// Device/Application/PLC_VISU
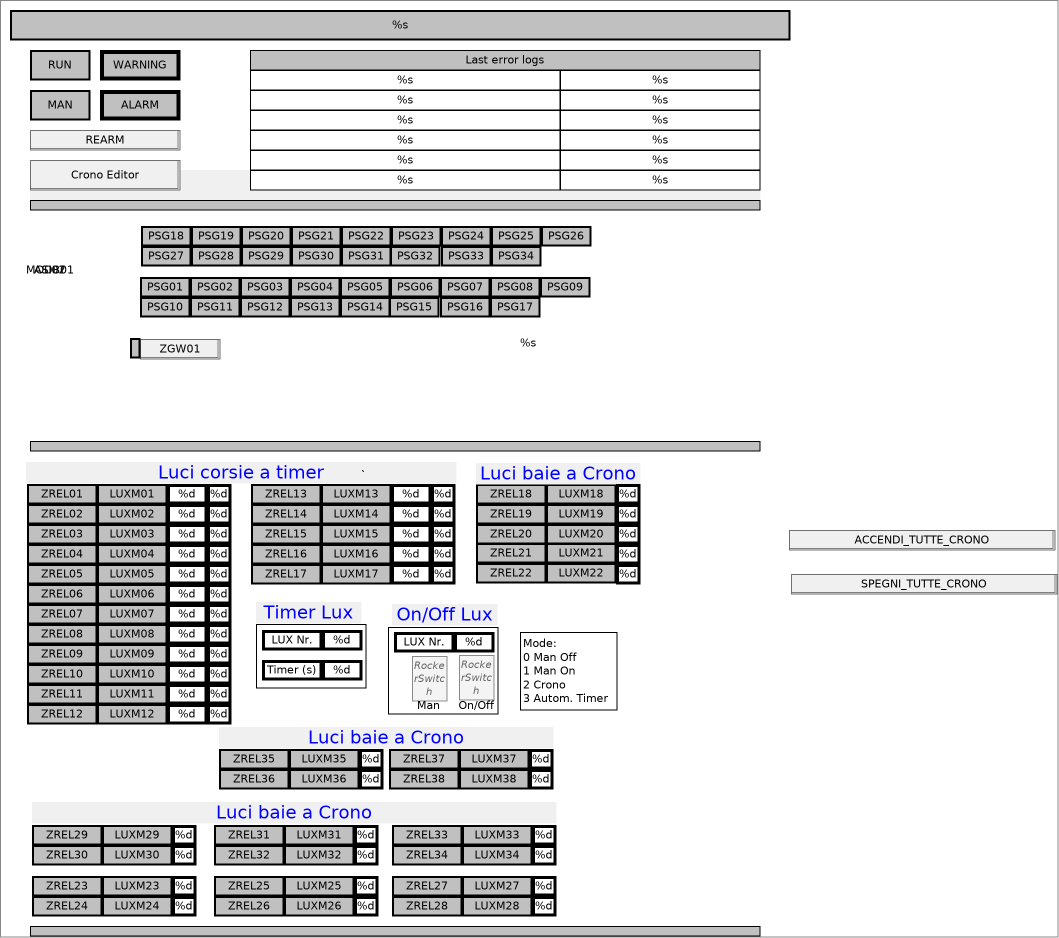
VISUALIZATION PLC_VISU  // 1059x938
    Rectangle (10,10 780x30), "%s", text variable: Plant_NAME
    Rectangle (30,441 730x10)
    Rectangle (30,170 730x30)
    Rectangle (30,926 730x10)
    Rectangle (30,200 730x10)
    Rectangle (319,333 220x20), "%s", text variable: Sys.Time_LogString
    Polygon (50,270), "MODB01", colour variable: MODB01.Status_Vis
    RoundedRectangle (30,50 60x30), "RUN", colour toggle: NOT Mode_Manual
        OnMouseUp: execute { Mode_Manual:=(FALSE); }
    RoundedRectangle (30,90 60x30), "MAN", colour toggle: Mode_Manual
        OnMouseUp: execute { Mode_Manual:=(TRUE); }
    Button (30,160 150x30), "Crono Editor"
        OnMouseUp:  Assign=VIS_CHONOEDITOR, Assign=VIS_CHONOEDITOR, Type=Assignment
    Rectangle (560,70 200x20), "%s", text variable: SYS.LastLogs_Msg[0]
    Polygon (240,190), invisible if: SYS.LastLogs_Idx<>0
    Rectangle (560,90 200x20), "%s", text variable: SYS.LastLogs_Msg[1]
    Polygon (240,90), invisible if: SYS.LastLogs_Idx<>1
    Rectangle (560,110 200x20), "%s", text variable: SYS.LastLogs_Msg[2]
    Polygon (240,110), invisible if: SYS.LastLogs_Idx<>2
    Rectangle (560,130 200x20), "%s", text variable: SYS.LastLogs_Msg[3]
    Polygon (240,130), invisible if: SYS.LastLogs_Idx<>3
    Rectangle (560,150 200x20), "%s", text variable: SYS.LastLogs_Msg[4]
    Polygon (240,150), invisible if: SYS.LastLogs_Idx<>4
    Rectangle (560,170 200x20), "%s", text variable: SYS.LastLogs_Msg[5]
    Polygon (240,170), invisible if: SYS.LastLogs_Idx<>5
    Rectangle (250,70 310x20), "%s", text variable: SYS.LastLogs_Dat[0]
    Rectangle (250,90 310x20), "%s", text variable: SYS.LastLogs_Dat[1]
    Rectangle (250,110 310x20), "%s", text variable: SYS.LastLogs_Dat[2]
    Rectangle (250,130 310x20), "%s", text variable: SYS.LastLogs_Dat[3]
    Rectangle (250,150 310x20), "%s", text variable: SYS.LastLogs_Dat[4]
    Rectangle (250,170 310x20), "%s", text variable: SYS.LastLogs_Dat[5]
    Rectangle (100,90 80x30), "ALARM", colour toggle: SYS.Alarm
    Rectangle (100,50 80x30), "WARNING", colour toggle: SYS.Warning
    Button (30,130 150x20), "REARM"
        OnMouseUp: execute { SYS.Alarm:=(FALSE); }
        OnMouseUp: execute { SYS.Warning:=(FALSE); }
    Rectangle (250,50 510x20), "Last error logs"
    Polygon (50,270), "ASI01", colour variable: ASI01.Status_Vis
    Polygon (50,270), "ASI02", colour variable: ASI02.Status_Vis
    Button (140,339 80x20), "ZGW01"
    Rectangle (130,338 10x20), colour variable: ZGW01.Status_Vis
    Line (130,246)
    Rectangle (140,297 50x20), "PSG10", colour variable: PSG[10].Status_Vis
    Rectangle (190,297 50x20), "PSG11", colour variable: PSG[11].Status_Vis
    Rectangle (240,297 50x20), "PSG12", colour variable: PSG[12].Status_Vis
    Rectangle (290,297 50x20), "PSG13", colour variable: PSG[13].Status_Vis
    Rectangle (219,769 70x20), "ZREL36", colour variable: ZREL[36].Status_Vis
    Rectangle (289,769 70x20), "LUXM36", colour variable: LUXM[36].Status_Vis
    Rectangle (219,749 70x20), "ZREL35", colour variable: ZREL[35].Status_Vis
    Rectangle (289,749 70x20), "LUXM35", colour variable: LUXM[35].Status_Vis
    Rectangle (389,769 70x20), "ZREL38", colour variable: ZREL[38].Status_Vis
    Rectangle (459,769 70x20), "LUXM38", colour variable: LUXM[38].Status_Vis
    Rectangle (389,749 70x20), "ZREL37", colour variable: ZREL[37].Status_Vis
    Rectangle (459,749 70x20), "LUXM37", colour variable: LUXM[37].Status_Vis
    Rectangle (219,727 334x21), "Luci baie a Crono"
    Rectangle (476,484 70x20), "ZREL18", colour variable: ZREL[18].Status_Vis
    Rectangle (476,504 70x20), "ZREL19", colour variable: ZREL[19].Status_Vis
    Rectangle (476,524 70x20), "ZREL20", colour variable: ZREL[20].Status_Vis
    Rectangle (476,543 70x20), "ZREL21", colour variable: ZREL[21].Status_Vis
    Rectangle (476,563 70x20), "ZREL22", colour variable: ZREL[22].Status_Vis
    Group (546,484 70x99)
        Rectangle (0,0 70x20), "LUXM18", colour variable: LUXM[18].Status_Vis
        Rectangle (0,20 70x20), "LUXM19", colour variable: LUXM[19].Status_Vis
        Rectangle (0,40 70x20), "LUXM20", colour variable: LUXM[20].Status_Vis
        Rectangle (0,59 70x20), "LUXM21", colour variable: LUXM[21].Status_Vis
        Rectangle (0,79 70x20), "LUXM22", colour variable: LUXM[22].Status_Vis
    Rectangle (476,463 164x21), "Luci baie a Crono"
    Rectangle (32,896 70x20), "ZREL24", colour variable: ZREL[24].Status_Vis
    Rectangle (102,896 70x20), "LUXM24", colour variable: LUXM[24].Status_Vis
    Rectangle (32,876 70x20), "ZREL23", colour variable: ZREL[23].Status_Vis
    Rectangle (102,876 70x20), "LUXM23", colour variable: LUXM[23].Status_Vis
    Rectangle (214,896 70x20), "ZREL26", colour variable: ZREL[26].Status_Vis
    Rectangle (284,896 70x20), "LUXM26", colour variable: LUXM[26].Status_Vis
    Rectangle (214,876 70x20), "ZREL25", colour variable: ZREL[25].Status_Vis
    Rectangle (284,876 70x20), "LUXM25", colour variable: LUXM[25].Status_Vis
    Rectangle (392,896 70x20), "ZREL28", colour variable: ZREL[28].Status_Vis
    Rectangle (462,896 70x20), "LUXM28", colour variable: LUXM[28].Status_Vis
    Rectangle (392,876 70x20), "ZREL27", colour variable: ZREL[27].Status_Vis
    Rectangle (462,876 70x20), "LUXM27", colour variable: LUXM[27].Status_Vis
    Rectangle (32,845 70x20), "ZREL30", colour variable: ZREL[30].Status_Vis
    Rectangle (102,845 70x20), "LUXM30", colour variable: LUXM[30].Status_Vis
    Rectangle (32,825 70x20), "ZREL29", colour variable: ZREL[29].Status_Vis
    Rectangle (102,825 70x20), "LUXM29", colour variable: LUXM[29].Status_Vis
    Rectangle (214,845 70x20), "ZREL32", colour variable: ZREL[32].Status_Vis
    Rectangle (284,845 70x20), "LUXM32", colour variable: LUXM[32].Status_Vis
    Rectangle (214,825 70x20), "ZREL31", colour variable: ZREL[31].Status_Vis
    Rectangle (284,825 70x20), "LUXM31", colour variable: LUXM[31].Status_Vis
    Rectangle (392,845 70x20), "ZREL34", colour variable: ZREL[34].Status_Vis
    Rectangle (462,845 70x20), "LUXM34", colour variable: LUXM[34].Status_Vis
    Rectangle (392,825 70x20), "ZREL33", colour variable: ZREL[33].Status_Vis
    Rectangle (462,825 70x20), "LUXM33", colour variable: LUXM[33].Status_Vis
    Rectangle (32,802 524x21), "Luci baie a Crono"
    Rectangle (340,297 50x20), "PSG14", colour variable: PSG[14].Status_Vis
    Rectangle (140,277 50x20), "PSG01", colour variable: PSG[1].Status_Vis
    Rectangle (190,277 50x20), "PSG02", colour variable: PSG[2].Status_Vis
    Rectangle (240,277 50x20), "PSG03", colour variable: PSG[3].Status_Vis
    Rectangle (290,277 50x20), "PSG04", colour variable: PSG[4].Status_Vis
    Rectangle (340,277 50x20), "PSG05", colour variable: PSG[5].Status_Vis
    Rectangle (390,277 50x20), "PSG06", colour variable: PSG[6].Status_Vis
    Rectangle (440,277 50x20), "PSG07", colour variable: PSG[7].Status_Vis
    Rectangle (490,277 50x20), "PSG08", colour variable: PSG[8].Status_Vis
    Rectangle (540,277 50x20), "PSG09", colour variable: PSG[9].Status_Vis
    Rectangle (389,297 50x20), "PSG15", colour variable: PSG[15].Status_Vis
    Rectangle (440,297 50x20), "PSG16", colour variable: PSG[16].Status_Vis
    Rectangle (490,297 50x20), "PSG17", colour variable: PSG[17].Status_Vis
    Rectangle (141,246 50x20), "PSG27", colour variable: PSG[27].Status_Vis
    Rectangle (191,246 50x20), "PSG28", colour variable: PSG[28].Status_Vis
    Rectangle (241,246 50x20), "PSG29", colour variable: PSG[29].Status_Vis
    Rectangle (291,246 50x20), "PSG30", colour variable: PSG[30].Status_Vis
    Rectangle (341,246 50x20), "PSG31", colour variable: PSG[31].Status_Vis
    Rectangle (141,226 50x20), "PSG18", colour variable: PSG[18].Status_Vis
    Rectangle (191,226 50x20), "PSG19", colour variable: PSG[19].Status_Vis
    Rectangle (241,226 50x20), "PSG20", colour variable: PSG[20].Status_Vis
    Rectangle (291,226 50x20), "PSG21", colour variable: PSG[21].Status_Vis
    Rectangle (341,226 50x20), "PSG22", colour variable: PSG[22].Status_Vis
    Rectangle (391,226 50x20), "PSG23", colour variable: PSG[23].Status_Vis
    Rectangle (441,226 50x20), "PSG24", colour variable: PSG[24].Status_Vis
    Rectangle (491,226 50x20), "PSG25", colour variable: PSG[25].Status_Vis
    Rectangle (541,226 50x20), "PSG26", colour variable: PSG[26].Status_Vis
    Rectangle (390,246 50x20), "PSG32", colour variable: PSG[32].Status_Vis
    Rectangle (441,246 50x20), "PSG33", colour variable: PSG[33].Status_Vis
    Rectangle (491,246 50x20), "PSG34", colour variable: PSG[34].Status_Vis
    Group (256,602 110x86)
        Rectangle (0,22 110x64)
        Rectangle (6,28 60x20), "LUX Nr."
        Rectangle (66,28 40x20), "%d", text variable: PLC_PRG.TimerLuxSelected
            OnMouseDown: write the text variable via Edit, min 1, max ACTIVELUX, title '1'
        Rectangle (66,58 40x20), "%d", text variable: LUXM[PLC_PRG.TimerLuxSelected].StrLuxTimer
            OnMouseDown: write the text variable via Edit, min 10, max 32760, title '1'
        Rectangle (6,58 60x20), "Timer (s)"
        Rectangle (0,0 105x21), "Timer Lux"
    Line (396,474) (396,474)
    Rectangle (26,462 430x21), "Luci corsie a timer"
    Rectangle (97,484 70x20), "LUXM01", colour variable: LUXM[1].Status_Vis
    Rectangle (27,484 70x20), "ZREL01", colour variable: ZREL[1].Status_Vis
    Rectangle (97,504 70x20), "LUXM02", colour variable: LUXM[2].Status_Vis
    Rectangle (27,504 70x20), "ZREL02", colour variable: ZREL[2].Status_Vis
    Rectangle (97,524 70x20), "LUXM03", colour variable: LUXM[3].Status_Vis
    Rectangle (27,524 70x20), "ZREL03", colour variable: ZREL[3].Status_Vis
    Rectangle (97,544 70x20), "LUXM04", colour variable: LUXM[4].Status_Vis
    Rectangle (27,544 70x20), "ZREL04", colour variable: ZREL[4].Status_Vis
    Rectangle (97,564 70x20), "LUXM05", colour variable: LUXM[5].Status_Vis
    Rectangle (27,564 70x20), "ZREL05", colour variable: ZREL[5].Status_Vis
    Rectangle (97,584 70x20), "LUXM06", colour variable: LUXM[6].Status_Vis
    Rectangle (27,584 70x20), "ZREL06", colour variable: ZREL[6].Status_Vis
    Rectangle (97,604 70x20), "LUXM07", colour variable: LUXM[7].Status_Vis
    Rectangle (27,604 70x20), "ZREL07", colour variable: ZREL[7].Status_Vis
    Rectangle (97,624 70x20), "LUXM08", colour variable: LUXM[8].Status_Vis
    Rectangle (27,624 70x20), "ZREL08", colour variable: ZREL[8].Status_Vis
    Rectangle (97,644 70x20), "LUXM09", colour variable: LUXM[9].Status_Vis
    Rectangle (27,644 70x20), "ZREL09", colour variable: ZREL[9].Status_Vis
    Rectangle (97,664 70x20), "LUXM10", colour variable: LUXM[10].Status_Vis
    Rectangle (27,664 70x20), "ZREL10", colour variable: ZREL[10].Status_Vis
    Rectangle (97,684 70x20), "LUXM11", colour variable: LUXM[11].Status_Vis
    Rectangle (27,684 70x20), "ZREL11", colour variable: ZREL[11].Status_Vis
    Rectangle (97,704 70x20), "LUXM12", colour variable: LUXM[12].Status_Vis
    Rectangle (27,704 70x20), "ZREL12", colour variable: ZREL[12].Status_Vis
    Rectangle (251,484 70x20), "ZREL13", colour variable: ZREL[13].Status_Vis
    Rectangle (321,484 70x20), "LUXM13", colour variable: LUXM[13].Status_Vis
    Rectangle (251,504 70x20), "ZREL14", colour variable: ZREL[14].Status_Vis
    Rectangle (321,504 70x20), "LUXM14", colour variable: LUXM[14].Status_Vis
    Rectangle (251,524 70x20), "ZREL15", colour variable: ZREL[15].Status_Vis
    Rectangle (321,524 70x20), "LUXM15", colour variable: LUXM[15].Status_Vis
    Rectangle (251,544 70x20), "ZREL16", colour variable: ZREL[16].Status_Vis
    Rectangle (321,544 70x20), "LUXM16", colour variable: LUXM[16].Status_Vis
    Rectangle (251,564 70x20), "ZREL17", colour variable: ZREL[17].Status_Vis
    Rectangle (321,564 70x20), "LUXM17", colour variable: LUXM[17].Status_Vis
    Polyline (362,470) (363,471)
    Rectangle (167,484 40x20), "%d", text variable: LUXM[1].StrLuxTimer, colour toggle: CronEd.CN_Sel<>CronEd.CN_Act
        OnMouseDown: write the text variable via Edit, min 10, max 32760, title '1'
    Rectangle (167,504 40x20), "%d", text variable: LUXM[2].StrLuxTimer, colour toggle: CronEd.CN_Sel<>CronEd.CN_Act
        OnMouseDown: write the text variable via Edit, min 10, max 32760, title '1'
    Rectangle (167,524 40x20), "%d", text variable: LUXM[3].StrLuxTimer, colour toggle: CronEd.CN_Sel<>CronEd.CN_Act
        OnMouseDown: write the text variable via Edit, min 10, max 32760, title '1'
    Rectangle (167,544 40x20), "%d", text variable: LUXM[4].StrLuxTimer, colour toggle: CronEd.CN_Sel<>CronEd.CN_Act
        OnMouseDown: write the text variable via Edit, min 10, max 32760, title '1'
    Rectangle (167,564 40x20), "%d", text variable: LUXM[5].StrLuxTimer, colour toggle: CronEd.CN_Sel<>CronEd.CN_Act
        OnMouseDown: write the text variable via Edit, min 10, max 32760, title '1'
    Rectangle (167,584 40x20), "%d", text variable: LUXM[6].StrLuxTimer, colour toggle: CronEd.CN_Sel<>CronEd.CN_Act
        OnMouseDown: write the text variable via Edit, min 10, max 32760, title '1'
    Rectangle (167,604 40x20), "%d", text variable: LUXM[7].StrLuxTimer, colour toggle: CronEd.CN_Sel<>CronEd.CN_Act
        OnMouseDown: write the text variable via Edit, min 10, max 32760, title '1'
    Rectangle (167,624 40x20), "%d", text variable: LUXM[8].StrLuxTimer, colour toggle: CronEd.CN_Sel<>CronEd.CN_Act
        OnMouseDown: write the text variable via Edit, min 10, max 32760, title '1'
    Rectangle (167,644 40x20), "%d", text variable: LUXM[9].StrLuxTimer, colour toggle: CronEd.CN_Sel<>CronEd.CN_Act
        OnMouseDown: write the text variable via Edit, min 10, max 32760, title '1'
    Rectangle (167,664 40x20), "%d", text variable: LUXM[10].StrLuxTimer, colour toggle: CronEd.CN_Sel<>CronEd.CN_Act
        OnMouseDown: write the text variable via Edit, min 10, max 32760, title '1'
    Rectangle (167,684 40x20), "%d", text variable: LUXM[11].StrLuxTimer, colour toggle: CronEd.CN_Sel<>CronEd.CN_Act
        OnMouseDown: write the text variable via Edit, min 10, max 32760, title '1'
    Rectangle (167,704 40x20), "%d", text variable: LUXM[12].StrLuxTimer, colour toggle: CronEd.CN_Sel<>CronEd.CN_Act
        OnMouseDown: write the text variable via Edit, min 10, max 32760, title '1'
    Rectangle (391,484 40x20), "%d", text variable: LUXM[13].StrLuxTimer, colour toggle: CronEd.CN_Sel<>CronEd.CN_Act
        OnMouseDown: write the text variable via Edit, min 10, max 32760, title '1'
    Rectangle (391,504 40x20), "%d", text variable: LUXM[14].StrLuxTimer, colour toggle: CronEd.CN_Sel<>CronEd.CN_Act
        OnMouseDown: write the text variable via Edit, min 10, max 32760, title '1'
    Rectangle (391,524 40x20), "%d", text variable: LUXM[15].StrLuxTimer, colour toggle: CronEd.CN_Sel<>CronEd.CN_Act
        OnMouseDown: write the text variable via Edit, min 10, max 32760, title '1'
    Rectangle (391,544 40x20), "%d", text variable: LUXM[16].StrLuxTimer, colour toggle: CronEd.CN_Sel<>CronEd.CN_Act
        OnMouseDown: write the text variable via Edit, min 10, max 32760, title '1'
    Rectangle (391,564 40x20), "%d", text variable: LUXM[17].StrLuxTimer, colour toggle: CronEd.CN_Sel<>CronEd.CN_Act
        OnMouseDown: write the text variable via Edit, min 10, max 32760, title '1'
    Group (388,604 110x114)
        Rectangle (0,23 110x87)
        RockerSwitch (24,52 35x45), variable: LUXM[PLC_PRG.LuxSelected].PressKeyVisuMan, behaviour: TOGGLE, style: Switch-RockerSwitch-Blue
        Rectangle (6,28 60x20), "LUX Nr."
        Rectangle (66,28 40x20), "%d", text variable: PLC_PRG.LuxSelected
            OnMouseDown: write the text variable via Edit, min 1, max LUXM_MAX, title '1'
        Rectangle (4,0 105x21), "On/Off Lux"
        RockerSwitch (71,51 35x45), variable: LUXM[PLC_PRG.LuxSelected].PressKeyVisuOn, behaviour: TOGGLE, style: Switch-RockerSwitch-Blue
        Label (21,89 39x25), "Man"
        Label (69,89 39x25), "On/Off"
    Rectangle (207,484 24x20), "%d", text variable: LUXM[1].ModeToServer, colour toggle: CronEd.CN_Sel<>CronEd.CN_Act
        OnMouseDown: write the text variable via Edit, min 10, max 32760, title '1'
    Rectangle (207,504 24x20), "%d", text variable: LUXM[2].ModeToServer, colour toggle: CronEd.CN_Sel<>CronEd.CN_Act
        OnMouseDown: write the text variable via Edit, min 10, max 32760, title '1'
    Rectangle (207,524 24x20), "%d", text variable: LUXM[3].ModeToServer, colour toggle: CronEd.CN_Sel<>CronEd.CN_Act
        OnMouseDown: write the text variable via Edit, min 10, max 32760, title '1'
    Rectangle (207,544 24x20), "%d", text variable: LUXM[4].ModeToServer, colour toggle: CronEd.CN_Sel<>CronEd.CN_Act
        OnMouseDown: write the text variable via Edit, min 10, max 32760, title '1'
    Rectangle (207,564 24x20), "%d", text variable: LUXM[5].ModeToServer, colour toggle: CronEd.CN_Sel<>CronEd.CN_Act
        OnMouseDown: write the text variable via Edit, min 10, max 32760, title '1'
    Rectangle (207,584 24x20), "%d", text variable: LUXM[6].ModeToServer, colour toggle: CronEd.CN_Sel<>CronEd.CN_Act
        OnMouseDown: write the text variable via Edit, min 10, max 32760, title '1'
    Rectangle (207,604 24x20), "%d", text variable: LUXM[7].ModeToServer, colour toggle: CronEd.CN_Sel<>CronEd.CN_Act
        OnMouseDown: write the text variable via Edit, min 10, max 32760, title '1'
    Rectangle (207,624 24x20), "%d", text variable: LUXM[8].ModeToServer, colour toggle: CronEd.CN_Sel<>CronEd.CN_Act
        OnMouseDown: write the text variable via Edit, min 10, max 32760, title '1'
    Rectangle (207,644 24x20), "%d", text variable: LUXM[9].ModeToServer, colour toggle: CronEd.CN_Sel<>CronEd.CN_Act
        OnMouseDown: write the text variable via Edit, min 10, max 32760, title '1'
    Rectangle (207,704 24x20), "%d", text variable: LUXM[12].ModeToServer, colour toggle: CronEd.CN_Sel<>CronEd.CN_Act
        OnMouseDown: write the text variable via Edit, min 10, max 32760, title '1'
    Rectangle (207,664 24x20), "%d", text variable: LUXM[10].ModeToServer, colour toggle: CronEd.CN_Sel<>CronEd.CN_Act
        OnMouseDown: write the text variable via Edit, min 10, max 32760, title '1'
    Rectangle (207,684 24x20), "%d", text variable: LUXM[11].ModeToServer, colour toggle: CronEd.CN_Sel<>CronEd.CN_Act
        OnMouseDown: write the text variable via Edit, min 10, max 32760, title '1'
    Rectangle (431,524 24x20), "%d", text variable: LUXM[15].ModeToServer, colour toggle: CronEd.CN_Sel<>CronEd.CN_Act
        OnMouseDown: write the text variable via Edit, min 10, max 32760, title '1'
    Rectangle (431,484 24x20), "%d", text variable: LUXM[13].ModeToServer, colour toggle: CronEd.CN_Sel<>CronEd.CN_Act
        OnMouseDown: write the text variable via Edit, min 10, max 32760, title '1'
    Rectangle (431,504 24x20), "%d", text variable: LUXM[14].ModeToServer, colour toggle: CronEd.CN_Sel<>CronEd.CN_Act
        OnMouseDown: write the text variable via Edit, min 10, max 32760, title '1'
    Rectangle (431,544 24x20), "%d", text variable: LUXM[16].ModeToServer, colour toggle: CronEd.CN_Sel<>CronEd.CN_Act
        OnMouseDown: write the text variable via Edit, min 10, max 32760, title '1'
    Rectangle (431,564 24x20), "%d", text variable: LUXM[17].ModeToServer, colour toggle: CronEd.CN_Sel<>CronEd.CN_Act
        OnMouseDown: write the text variable via Edit, min 10, max 32760, title '1'
    Rectangle (616,484 24x20), "%d", text variable: LUXM[18].ModeToServer, colour toggle: CronEd.CN_Sel<>CronEd.CN_Act
        OnMouseDown: write the text variable via Edit, min 10, max 32760, title '1'
    Rectangle (616,504 24x20), "%d", text variable: LUXM[19].ModeToServer, colour toggle: CronEd.CN_Sel<>CronEd.CN_Act
        OnMouseDown: write the text variable via Edit, min 10, max 32760, title '1'
    Rectangle (616,524 24x20), "%d", text variable: LUXM[20].ModeToServer, colour toggle: CronEd.CN_Sel<>CronEd.CN_Act
        OnMouseDown: write the text variable via Edit, min 10, max 32760, title '1'
    Rectangle (616,564 24x20), "%d", text variable: LUXM[22].ModeToServer, colour toggle: CronEd.CN_Sel<>CronEd.CN_Act
        OnMouseDown: write the text variable via Edit, min 10, max 32760, title '1'
    Rectangle (616,544 24x20), "%d", text variable: LUXM[21].ModeToServer, colour toggle: CronEd.CN_Sel<>CronEd.CN_Act
        OnMouseDown: write the text variable via Edit, min 10, max 32760, title '1'
    Rectangle (359,749 24x20), "%d", text variable: LUXM[35].ModeToServer, colour toggle: CronEd.CN_Sel<>CronEd.CN_Act
        OnMouseDown: write the text variable via Edit, min 10, max 32760, title '1'
    Rectangle (359,769 24x20), "%d", text variable: LUXM[36].ModeToServer, colour toggle: CronEd.CN_Sel<>CronEd.CN_Act
        OnMouseDown: write the text variable via Edit, min 10, max 32760, title '1'
    Rectangle (172,845 24x20), "%d", text variable: LUXM[30].ModeToServer, colour toggle: CronEd.CN_Sel<>CronEd.CN_Act
        OnMouseDown: write the text variable via Edit, min 10, max 32760, title '1'
    Rectangle (172,825 24x20), "%d", text variable: LUXM[29].ModeToServer, colour toggle: CronEd.CN_Sel<>CronEd.CN_Act
        OnMouseDown: write the text variable via Edit, min 10, max 32760, title '1'
    Rectangle (529,749 24x20), "%d", text variable: LUXM[37].ModeToServer, colour toggle: CronEd.CN_Sel<>CronEd.CN_Act
        OnMouseDown: write the text variable via Edit, min 10, max 32760, title '1'
    Rectangle (529,769 24x20), "%d", text variable: LUXM[38].ModeToServer, colour toggle: CronEd.CN_Sel<>CronEd.CN_Act
        OnMouseDown: write the text variable via Edit, min 10, max 32760, title '1'
    Rectangle (172,896 24x20), "%d", text variable: LUXM[24].ModeToServer, colour toggle: CronEd.CN_Sel<>CronEd.CN_Act
        OnMouseDown: write the text variable via Edit, min 10, max 32760, title '1'
    Rectangle (172,876 24x20), "%d", text variable: LUXM[23].ModeToServer, colour toggle: CronEd.CN_Sel<>CronEd.CN_Act
        OnMouseDown: write the text variable via Edit, min 10, max 32760, title '1'
    Rectangle (354,845 24x20), "%d", text variable: LUXM[32].ModeToServer, colour toggle: CronEd.CN_Sel<>CronEd.CN_Act
        OnMouseDown: write the text variable via Edit, min 10, max 32760, title '1'
    Rectangle (354,825 24x20), "%d", text variable: LUXM[31].ModeToServer, colour toggle: CronEd.CN_Sel<>CronEd.CN_Act
        OnMouseDown: write the text variable via Edit, min 10, max 32760, title '1'
    Rectangle (354,896 24x20), "%d", text variable: LUXM[26].ModeToServer, colour toggle: CronEd.CN_Sel<>CronEd.CN_Act
        OnMouseDown: write the text variable via Edit, min 10, max 32760, title '1'
    Rectangle (354,876 24x20), "%d", text variable: LUXM[25].ModeToServer, colour toggle: CronEd.CN_Sel<>CronEd.CN_Act
        OnMouseDown: write the text variable via Edit, min 10, max 32760, title '1'
    Rectangle (532,896 24x20), "%d", text variable: LUXM[28].ModeToServer, colour toggle: CronEd.CN_Sel<>CronEd.CN_Act
        OnMouseDown: write the text variable via Edit, min 10, max 32760, title '1'
    Rectangle (532,876 24x20), "%d", text variable: LUXM[27].ModeToServer, colour toggle: CronEd.CN_Sel<>CronEd.CN_Act
        OnMouseDown: write the text variable via Edit, min 10, max 32760, title '1'
    Rectangle (532,845 24x20), "%d", text variable: LUXM[34].ModeToServer, colour toggle: CronEd.CN_Sel<>CronEd.CN_Act
        OnMouseDown: write the text variable via Edit, min 10, max 32760, title '1'
    Rectangle (532,825 24x20), "%d", text variable: LUXM[33].ModeToServer, colour toggle: CronEd.CN_Sel<>CronEd.CN_Act
        OnMouseDown: write the text variable via Edit, min 10, max 32760, title '1'
    Rectangle (520,632 97x78), "Mode: 0 Man Off 1 Man On 2 Crono 3 Autom. Timer"
    Button (789,530 266x20), "ACCENDI_TUTTE_CRONO"
        toggle testCronoOn
    Button (791,574 266x20), "SPEGNI_TUTTE_CRONO"
        toggle testCronoOff
END_VISUALIZATION
